TYPE ST_StationEvents :
STRUCT
	
	aEvents								: ARRAY [0..100] OF ST_EVENT;	
	
	bImmediateFault						: BOOL;
	bCycleStopFault						: BOOL;
	bCycleStopRequest					: BOOL;
			
END_STRUCT
END_TYPE

(* stored: Version 1.1.0.1, ProductVersion 3.1.4024.13
   DUT ST_StationEvents: Id {57187980-fadb-46c4-ba60-74da2804cdd1} *)
